(* IEC 61131-3 sources: embox/project/plc/matiec/lib/led, 1 file *)

(* ---- led.iecst ---- *)
FUNCTION_BLOCK LED_ON
VAR_INPUT
LED: UINT;
END_VAR
VAR_OUTPUT
SUCCESS: BOOL;
END_VAR

  SUCCESS := 0;

END_FUNCTION_BLOCK

FUNCTION_BLOCK LED_OFF
VAR_INPUT
LED: UINT;
END_VAR
VAR_OUTPUT
SUCCESS: BOOL;
END_VAR

  SUCCESS := 0;

END_FUNCTION_BLOCK
